PROGRAM prgCom
VAR
	fbCom			: FB_MqttCommunicator;
END_VAR

fbCom(
	bConnect:= TRUE, 
	sUserName:= 'dd42716e-193d-4c6c-a2c4-46c477e1877b', 
	sUserPassword:= 'b13d7ac3-0642-4711-8449-ebfd8a27b319', 
	eSavePositionCertificate:= eSavePositionOnPLC.ePostionC, 
	bConnected=> , 
	bError=> , 
	hrErrorCode=> , 
	eConnectionState=> , 
	eErrorMessage_Out=> );

END_PROGRAM

(* stored: Version 1.1.0.1, ProductVersion 3.1.4024.11
   POU prgCom: Id {ab2e2113-e5ef-4576-b3e1-d9e4709b48fc}, SpecialFunc None *)
